Staubli VAL3: cycle_lock.pgx

program cycle_lock()
begin
  //
  // Lock by PLC THE CYCLE
  //
  if !cycleStatus:bPausePLC
    logMsg("[KERNEL] PLC:Lock the cycle")
    // lock it
    cycleStatus:bPausePLC=true
    stopMove()
    call OnEvent:OnCycleEvent(2)
    //
  endIf
  //
end
